FUNCTION_BLOCK FB_ACTransferControl
(*
Version history:
DATE		|	Version/Author 		|	Remark
----------------------------------------------------------------------------------------------------
16.03.12	|	2.000.001	PSA		|	Original Version.
									|	Runs Transfer Control.  
									|	Transfers Outers from the infeed conveyor to the lowerator.
*)
VAR_INPUT
	bTransferEnabled				: BOOL;						(* This block is active *)
	bMotorFault						: BOOL;						(* physical Drive fault input *)
	bPackPresent					: BOOL;						(* Pack is present and ready to transfer *)
	bExitBlocked					: BOOL;						(* Exit is blocked *)
	bDelayStop						: BOOL;						(* *)
	nRunSpeed						: WORD;						(* Set speed for the transfer motor *)
	fConversionFactor				: LREAL;					(* Converstion factor *)
	fPackPresentFilterTime			: LREAL;					(* Filter time for a pack to be present *)
	fExitBlockedFilterTime			: LREAL;					(* Filter time for the exit to be blocked *)
	nScalingFactor					: INT;						(* Scaling factor for the output *)
END_VAR
VAR_OUTPUT
	bTransferRun					: BOOL;
	nMotorAnalogueOutputSpeed		: UINT;
END_VAR
VAR
	bPackPresentFilter				: BOOL;
	bExitBlockedFilter				: BOOL;
	fbPackPresentTimer				: TON;
	fbExitBlockedTimer				: TON;
END_VAR

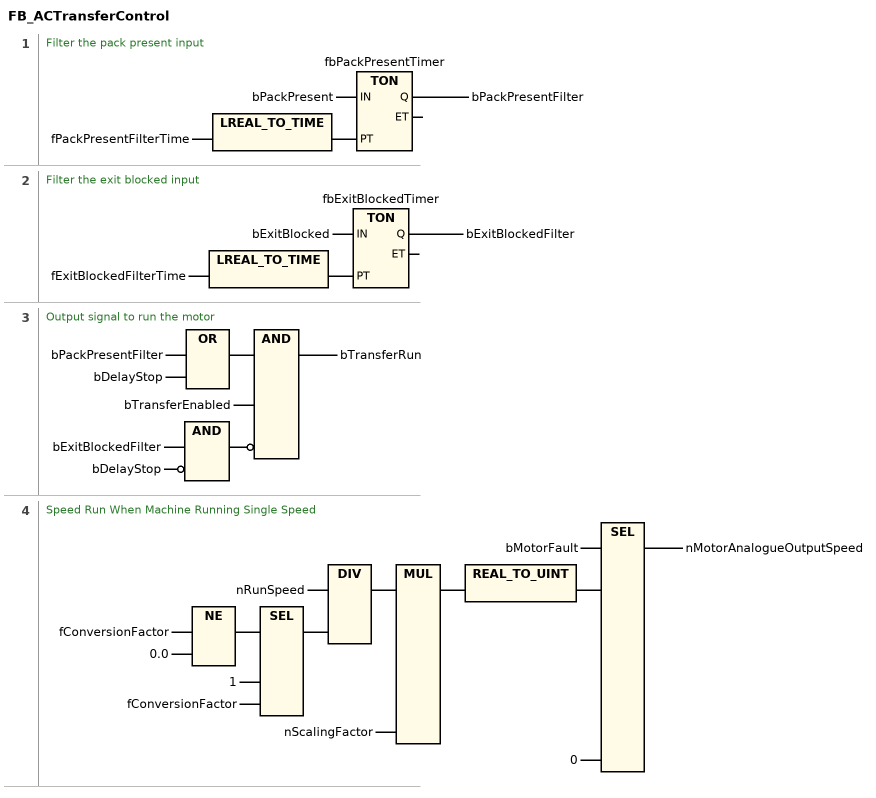
// NETWORK 1
// Filter the pack present input
fbPackPresentTimer(IN := bPackPresent, PT := LREAL_TO_TIME(fPackPresentFilterTime)); // TON
bPackPresentFilter := fbPackPresentTimer.Q;

// NETWORK 2
// Filter the exit blocked input
fbExitBlockedTimer(IN := bExitBlocked, PT := LREAL_TO_TIME(fExitBlockedFilterTime)); // TON
bExitBlockedFilter := fbExitBlockedTimer.Q;

// NETWORK 3
// Output signal to run the motor
bTransferRun := (bPackPresentFilter OR bDelayStop) AND bTransferEnabled AND NOT (bExitBlockedFilter AND NOT bDelayStop);

// NETWORK 4
// Speed Run When Machine Running Single Speed
nMotorAnalogueOutputSpeed := SEL(bMotorFault, REAL_TO_UINT((nRunSpeed / SEL(fConversionFactor <> 0.0, 1, fConversionFactor)) * nScalingFactor), 0);

END_FUNCTION_BLOCK

(* stored: Version 1.1.0.1, ProductVersion 3.1.4024.15
   POU FB_ACTransferControl: Id {8802ce64-56a7-44ad-8618-df389d32fc69}, SpecialFunc None *)
